PROGRAM MAIN

flyingsaw.Master();
flyingsaw.Slave();

flyingsaw.checkPower();
flyingsaw.checkFlyingSaw();
flyingsaw.checkMove();
flyingsaw.checkReset();

END_PROGRAM

(* stored: Version 1.1.0.1, ProductVersion 3.1.4024.4
   POU MAIN: Id {7f83cc0a-42dc-414a-a914-ff841541d6be}, SpecialFunc None *)
